// TwinCAT 3 PLC project SCARAFITTI
// ProgramVersion: 3.1.4023.0
// libraries:
//   Tc2_ControllerToolbox, * (Beckhoff Automation GmbH)
//   Tc2_Standard, * (Beckhoff Automation GmbH)
//   Tc2_System, * (Beckhoff Automation GmbH)
//   Tc2_Utilities, * (Beckhoff Automation GmbH)
//   Tc3_Module, * (Beckhoff Automation GmbH)
//   VisuSymbols,3.5.10.0,System
// project tree:
//   / GlobalTextList.TcGTLO, PlcTask.TcTTO, FastTask.TcTTO
//   GVLs/ Diagrama.TcCD (not stored), Cilindro.TcDUT, GVL.TcGVL, IO.TcGVL, SCARAFITTI.TcDUT
//   POUs/Actuadores/ PWM_valvulas.TcPOU (not stored)
//   POUs/Comunicacion/ EjecutarComando.TcPOU, G_buscar_numero.TcPOU, InterpretarComando.TcPOU, LetraPresente.TcPOU
//   POUs/ FB_BARRIDOXY.TcPOU, FB_SOLVEABCDE.TcPOU, FB_SOLVEALFABETA.TcPOU, MAIN.TcPOU, Simulacion.TcPOU
//   POUs/Functions/ TwoPiCrop.TcPOU
//   POUs/Sensores/ EncoderMeas.TcPOU, ENCODERPULSEtoANGLE.TcPOU
// real-time tasks:
//   TASK PlcTask: cycle T#10ms, priority 20, ADS port 350
//   TASK FastTask: cycle T#1ms, priority 1, ADS port 351
//   TASK VISU_TASK: cycle T#200000us, priority 30, ADS port 352
// I/O:
//   DEVICE Device 1 (EtherCAT) (disabled), AmsNetId 172.17.69.129.2.1
//     Term 7 (EK1200) [EK1200-5000 EtherCAT Power supply (2A E-Bus)]
//       Term 8 (EL1004) [EL1004 4Ch. Dig. Input 24V, 3ms]
//       Term 9 (EL1004) [EL1004 4Ch. Dig. Input 24V, 3ms]
//       Term 10 (EL2004) [EL2004 4Ch. Dig. Output 24V, 0.5A]
//       Term 11 (EL2004) [EL2004 4Ch. Dig. Output 24V, 0.5A]
//       Term 13 (EL9011) [EL9011 End Terminal]
// variable links:
//   SCARAFITTI/SCARAFITTI Instance <-> Device 1 (EtherCAT)/Term 7 (EK1200)/Term 10 (EL2004)
//     FastTask Outputs/IO.valv_alfa_mas <-> Channel 1/Output
//     FastTask Outputs/IO.valv_alfa_menos <-> Channel 2/Output
//     FastTask Outputs/IO.valv_beta_mas <-> Channel 3/Output
//     FastTask Outputs/IO.valv_beta_menos <-> Channel 4/Output
//   SCARAFITTI/SCARAFITTI Instance <-> Device 1 (EtherCAT)/Term 7 (EK1200)/Term 9 (EL1004)
//     FastTask Inputs/IO.encoder1_A <-> Channel 1/Input
//     FastTask Inputs/IO.encoder1_B <-> Channel 2/Input

CONFIGURATION SCARAFITTI
    RESOURCE PLC ON TwinCAT3
        TASK PlcTask(INTERVAL := T#10ms, PRIORITY := 20);
        TASK FastTask(INTERVAL := T#1ms, PRIORITY := 1);
        PROGRAM MAIN WITH PlcTask : MAIN;
        PROGRAM Simulacion WITH PlcTask : Simulacion;
        PROGRAM EncoderMeas WITH FastTask : EncoderMeas;
        PROGRAM PWM_valvulas WITH FastTask : PWM_valvulas;
        PROGRAM Simulacion WITH FastTask : Simulacion;
    END_RESOURCE
END_CONFIGURATION

// ---- GVLs/Cilindro.TcDUT
TYPE Cilindro :
STRUCT
	posicion : REAL;
	extendido: BOOL;
	retraido: BOOL;
	parado: BOOL;
	extendiendo : BOOL;
	retrayendo: BOOL;
	regimen : REAL; //tnato por uno de apertura de válvula
END_STRUCT
END_TYPE

// ---- GVLs/SCARAFITTI.TcDUT
TYPE SCARAFITTI :
STRUCT
	parada : BOOL;
	simulacion_alfa : BOOL;
	simulacion_beta : BOOL;
	quieto : BOOL;
	en_objetivo : BOOL;
	error_objetivo : BOOL;
	ADSCOM_ready : BOOL;
END_STRUCT
END_TYPE

// ---- GVLs/GVL.TcGVL
{attribute 'qualified_only'}
VAR_GLOBAL


// Geometría del robot//
//todo en mm//

Pi : REAL := 3.1416;

d : REAL := 400;
l1 : REAL := 1000; //longitud brazo proximal
l2 : REAL := 1400; //longitud brazo distal

//Vértices robot

Xa : REAL:= 0; 
Ya : REAL:= 0; 
Xb : REAL:= 0; 
Yb : REAL:= 0; 
Xc : REAL:= 0; //posición x del spray
Xc_sp : REAL:= 0; //setpoint posición x del spray
Yc : REAL:= 0; //posición y del spray
Yc_sp : REAL:= 0; //setpoint posición y del spray
Xd : REAL:= 0; 
Yd : REAL:= 0; 
Xe : REAL:= 0; 
Ye : REAL:= 0; 

//Mitad de cada brazo

Xab : REAL:= 0; 
Yab : REAL:= 0; 
Xbc : REAL:= 0; 
Ybc : REAL:= 0; 
Xcd : REAL:= 0; 
Ycd : REAL:= 0; 
Xde : REAL:= 0; 
Yde : REAL:= 0;


//Ángulos

alfa : REAL:= 0; //ángulo del brazo proximal izquierdo
alfa_sp : REAL:= 0; //setpoint ángulo del brazo proximal izquierdo
beta : REAL:= 0; //ángulo del brazo proximal derecho
beta_sp: REAL:= 0; //setpoint ángulo del brazo proximal derecho

deadband_angulo : REAL:= 0.05; //banda de no actuación en torno a target [rad]

alfa1 : REAL:= 0; 
beta1 : REAL:= 0; 
alfa2 : REAL:= 0; 
beta2 : REAL:= 0; 


d1: REAL;
d2: REAL;


alfa_enc : REAL :=0;
beta_enc : REAL :=0;

//cilindros
Cilindro1 : Cilindro;
Cilindro2 : Cilindro;
regimen_maximo : REAL :=100;

//Internas
en_objetivo_alfa : BOOL; //brazo proximal izquierdo en posición objetivo
en_objetivo_beta : BOOL; ///brazo proximal derecho en posición objetivo
comando_actual : STRING := 'Default comando actual';
ultimo_comando : STRING;
comando_actual_tipo : STRING;

//Sistema
Scarafitti : SCARAFITTI;

END_VAR

// ---- GVLs/IO.TcGVL
{attribute 'qualified_only'}
VAR_GLOBAL
//INPUTS	
	encoder1_A AT %I* : BOOL;
	encoder1_B AT %I* : BOOL;
	encoder2_A AT %I* : BOOL;
	encoder2_B AT %I* : BOOL;
	tope_alfa AT %I* : BOOL;
	tope_beta AT %I* : BOOL;
	
// INPUTS SIMULACION
	alfa_sim : REAL:= GVL.Pi;
	beta_sim : REAL;
	
// INPUTS ADS
	string_in : STRING := 'Default command PC-PLC';
	string_out : STRING:= 'Default feedback PLC-PC';
	
//OUTPUTS	
	blink AT %Q* : BOOL := 1;
	valv_alfa_mas AT %Q* : BOOL;
	valv_alfa_menos AT %Q* : BOOL;
	valv_beta_mas AT %Q* : BOOL;
	valv_beta_menos AT %Q* : BOOL;	
	
//OUTPUTS ADS
	Xc_ADS : INT;
	Yc_ADS : INT;
	alfa_deg:REAL;
	beta_deg:REAL;
END_VAR

// ---- POUs/MAIN.TcPOU
PROGRAM MAIN
VAR
	
fb_solveAlfaBeta:FB_SOLVEALFABETA;
fb_solveABCDE:FB_SOLVEABCDE;
fb_barridoXY:FB_BARRIDOXY;
InterpretarComando : InterpretarComando;
EjecutarComando: EjecutarComando;




Xc_test : LINT;
aux_ADS : INT;
Yc_test : LINT;

//test
nVar: UDINT;
//test
aux_UDINT : UDINT;
aux_REAL : REAL;

END_VAR

//Blink
IO.blink := NOT(IO.blink);


//DÓNDE ESTOY?
///comunicar ángulos
IO.alfa_deg:=GVL.alfa*180/GVL.Pi;
IO.beta_deg:=GVL.beta*180/GVL.Pi;
///Resolver geometría
////SolveABCDE
fb_solveABCDE.alfa:=GVL.alfa;
fb_solveABCDE.beta:=GVL.beta;
fb_solveABCDE();
GVL.Xa:=(fb_solveABCDE.Xa);
GVL.Ya:=(fb_solveABCDE.Ya);
GVL.Xb:=(fb_solveABCDE.Xb);
GVL.Yb:=(fb_solveABCDE.Yb);
GVL.Xc:=(fb_solveABCDE.Xc);
IO.Xc_ADS:=REAL_TO_INT(GVL.Xc);
IO.Yc_ADS:=REAL_TO_INT(GVL.Yc);
GVL.Yc:=(fb_solveABCDE.Yc);
GVL.Xd:=(fb_solveABCDE.Xd);
GVL.Yd:=(fb_solveABCDE.Yd);
GVL.Xe:=(fb_solveABCDE.Xe);
GVL.Ye:=(fb_solveABCDE.Ye);
////Brazos
GVL.Xab:=(GVL.Xa+GVL.Xb)/2;
GVL.Yab:=(GVL.Ya+GVL.Yb)/2;
GVL.Xbc:=(GVL.Xc+GVL.Xb)/2;
GVL.Ybc:=(GVL.Yc+GVL.Yb)/2;
GVL.Xcd:=(GVL.Xc+GVL.Xd)/2;
GVL.Ycd:=(GVL.Yc+GVL.Yd)/2;
GVL.Xde:=(GVL.Xd+GVL.Xe)/2;
GVL.Yde:=(GVL.Yd+GVL.Ye)/2;

//ADÓNDE VOY?
///Consigna XcYc
////Barrido para test
//fb_barridoXY.speed:=2;
//fb_barridoXY();
//GVL.Xc_sp:=fb_barridoXY.Xbarrido;
//GVL.Yc_sp:=fb_barridoXY.Ybarrido;
////ADS Com
IF ((NOT(GVL.Scarafitti.parada) AND GVL.Scarafitti.ADSCOM_ready AND IO.string_in<>GVL.ultimo_comando)OR IO.string_in='reset') THEN
	InterpretarComando();
	ELSE
		////Ignorar comandos que llegan mientras ADS com no está listo
		IO.string_in:=GVL.ultimo_comando;
END_IF

	

////Fija
//GVL.Xc_sp:= Xc_test;
//GVL.Yc_sp:= Yc_test;
///SolveAlfaBeta_sp
fb_solveAlfaBeta.x:=GVL.Xc_sp;
fb_solveAlfaBeta.y:=GVL.Yc_sp;
fb_solveAlfaBeta();
GVL.d1 :=fb_solveAlfaBeta.d1;
GVL.d2 :=fb_solveAlfaBeta.d2;
GVL.Scarafitti.error_objetivo := fb_solveAlfaBeta.error;
GVL.alfa_sp:=MIN(MAX(gvl.pi/2,fb_solveAlfaBeta.alfa),GVL.Pi);
GVL.beta_sp:=MIN(MAX(0,fb_solveAlfaBeta.beta),GVL.Pi/2);

//HE LLEGADO?
GVL.en_objetivo_alfa:=(ABS(GVL.alfa-GVL.alfa_sp)<=GVL.deadband_angulo);
GVL.en_objetivo_beta:=(ABS(GVL.beta-GVL.beta_sp)<=GVL.deadband_angulo);
GVL.Scarafitti.en_objetivo := GVL.en_objetivo_alfa AND GVL.en_objetivo_beta;


//SI NO HE LLEGADO, ME MUEVO
///si no hay parada
EjecutarComando();

END_PROGRAM

// ---- POUs/FB_SOLVEALFABETA.TcPOU
FUNCTION_BLOCK FB_SOLVEALFABETA
VAR_INPUT
x : REAL;
y : REAL;
END_VAR
VAR_OUTPUT
alfa : REAL;
beta : REAL;
d1 : REAL;
d2 : REAL;
alfa1 : REAL;
alfa2 : REAL;
beta1 : REAL;
beta2 : REAL;
error: BOOL := 0;

END_VAR
VAR
END_VAR

error:=FALSE;
d1 := SQRT(y*y+(x+GVL.d)*(x+GVL.d));
IF d1>(GVL.l1*GVL.l1+GVL.l2*GVL.l2) THEN
	error:=TRUE;
END_IF
d2 := SQRT(y*y+(x-GVL.d)*(x-GVL.d));
IF d2>(GVL.l1*GVL.l1+GVL.l2*GVL.l2) THEN
	error:=TRUE;
END_IF

IF (x+GVL.d=0) THEN
	alfa1:=GVL.Pi/2;
	ELSE IF x+GVL.d<0 THEN		
		alfa1 := gvl.pi + ATAN (y/(x+GVL.d));
		ELSE
			alfa1 := ATAN (y/(x+GVL.d));
		END_IF
	END_IF
IF alfa1 < 0 THEN
	error:=TRUE;
END_IF

IF (x-GVL.d=0) THEN
	beta1:=GVL.Pi/2;
	ELSE IF x-GVL.d>0 THEN
		beta1 := ATAN (y/(x-GVL.d));
	ELSE
		beta1 := GVL.Pi	+ ATAN (y/(x-GVL.d));
	END_IF
	END_IF

IF beta1 < 0 THEN
	error:=TRUE;
END_IF

IF (ABS((GVL.l1*GVL.l1+d1*d1-GVL.l2*GVL.l2)/(2*GVL.l1*d1))>1) THEN
error := TRUE;
END_IF

IF (ABS((GVL.l1*GVL.l1+d2*d2-GVL.l2*GVL.l2)/(2*GVL.l1*d2))>1) THEN
error := TRUE;
END_IF

IF error=FALSE THEN
	IF d1=0 THEN
		alfa2:=0;
		ELSE
			alfa2 := ABS(ACOS((GVL.l1*GVL.l1+d1*d1-GVL.l2*GVL.l2)/(2*GVL.l1*d1)));
		END_IF

	
	IF d2=0 THEN
		beta2:=0;
		ELSE
			beta2 := ABS(ACOS((GVL.l1*GVL.l1+d2*d2-GVL.l2*GVL.l2)/(2*GVL.l1*d2)));
		END_IF
alfa := alfa1 + alfa2;
beta := beta1 - beta2;
	END_IF

END_FUNCTION_BLOCK

// ---- POUs/FB_SOLVEABCDE.TcPOU
FUNCTION_BLOCK FB_SOLVEABCDE
VAR_INPUT
	alfa : REAL:= 0; //ángulo del brazo pxosimal izquierdo
	beta : REAL:= 0; //ángulo del brazo pxosimal derecho
END_VAR
VAR_OUTPUT
	
	Xa : REAL:= 0; 
	Ya : REAL:= 0; 
	Xb : REAL:= 0; 
	Yb : REAL:= 0; 
	Xc : REAL:= 0; 
	Yc : REAL:= 0;
	Xd : REAL:= 0; 
	Yd : REAL:= 0; 
	Xe : REAL:= 0; 
	Ye : REAL:= 0; 
	error : BOOL :=0;
	check_AB : REAL:=GVL.l1;
	check_BC : REAL:=GVL.l2;
	check_CD : REAL:=GVL.l2;
	check_DE : REAL:=GVL.l1;
	

END_VAR
VAR
	aux1 : REAL;
	aux2 : REAL;
	A : REAL;
	B : REAL;
	C : REAL;
END_VAR

error:=FALSE;

// A
Xa := -GVL.d ;
Ya := 0 ;

//B
Xb := Xa + GVL.l1*COS(alfa);
Yb := GVL.l1*SIN(alfa);

//E
Xe := GVL.d ;
Ye := 0 ;

//D
Xd := Xe + GVL.l1*COS(beta);
Yd := GVL.l1*SIN(beta);

//Chekcs
IF SQRT((Xd-Xb)*(Xd-Xb)+(Yd-Yb)*(Yd-Yb))>2*GVL.l2 THEN //B y D demaisado separados
	error:=TRUE;
	ELSE IF Xb>=Xd THEN //brazos proximales cruzados
		error:=TRUE;
		ELSE //calculate Xc
			aux1:=(Xb*Xb-Xd*Xd+Yb*Yb-Yd*Yd)/(2*(Xb-Xd));
			aux2:=-(Yb-Yd)/(Xb-Xd);
			A:=1+ aux2*aux2 ;
			B:=2*(aux1*aux2-Xb*aux2-Yb);
			C:=aux1*aux1-2*Xb*aux1+Yb*Yb+Xb*Xb-GVL.l2*GVL.l2;
			Yc := (-B+SQRT(B*B-4*A*C))/(2*A);
			Xc := aux1+aux2*Yc;
		END_IF
		
check_AB:=SQRT((Xb-Xa)*(Xb-Xa)+(Yb-Ya)*(Yb-Ya));
check_BC:=SQRT((Xb-Xc)*(Xb-Xc)+(Yb-Yc)*(Yb-Yc));
check_CD:=SQRT((Xd-Xc)*(Xd-Xc)+(Yd-Yc)*(Yd-Yc));
check_DE:=SQRT((Xd-Xe)*(Xd-Xe)+(Yd-Ye)*(Yd-Ye));
		
	END_IF

END_FUNCTION_BLOCK

// ---- POUs/FB_BARRIDOXY.TcPOU
FUNCTION_BLOCK FB_BARRIDOXY
VAR_INPUT
	speed : REAL;
END_VAR
VAR_OUTPUT
	Xbarrido: REAL := 0;
	Ybarrido : REAL :=1000;
END_VAR
VAR
	xmax : REAL := 500;
	ymin : REAL := 500;
	ymax : REAL := 1500;
	fase : INT := 1;
END_VAR

CASE fase OF
	1:
	IF Xbarrido + speed > xmax THEN
		fase:=2;
		ELSE
			Xbarrido := Xbarrido + speed;
	END_IF
	2:
	IF Ybarrido + speed > ymax THEN
		fase:=3;
		ELSE
			Ybarrido := Ybarrido + speed;
	END_IF
	3:
	IF Xbarrido - speed < -xmax THEN
		fase:=4;
		ELSE
			Xbarrido := Xbarrido - speed;
	END_IF
	4:
	IF Ybarrido - speed < ymin THEN
		fase:=1;
		ELSE
			Ybarrido := Ybarrido - speed;
	END_IF
END_CASE

END_FUNCTION_BLOCK

// ---- POUs/Comunicacion/InterpretarComando.TcPOU
FUNCTION_BLOCK InterpretarComando
VAR_INPUT
END_VAR
VAR_OUTPUT
	comando_valido:BOOL;
END_VAR
VAR
	aux_str:STRING;
	aux_int:INT;
	aux_real:REAL;
	buscarX:G_buscar_numero;
	buscarY:G_buscar_numero;
	buscarF:G_buscar_numero;
	buscarS:G_buscar_numero;
	
END_VAR

comando_valido:=FALSE;
///Comando en mayúsculas
IO.string_in:=f_toucase(IO.string_in);
///excepcion para reset
IF IO.string_in='RESET' THEN
	IO.string_in:='G00 X000 Y000';
END_IF
	IF  letraPresente('G',IO.string_in) THEN
		IF letraPresente('G00',IO.string_in) THEN
			IO.string_out:='comando G00 recibido';
			//buscar comandos de X
			IF letraPresente('X',IO.string_in) THEN
			buscarX.cadena:=IO.string_in;
			buscarX.letra:='X';
			buscarX();
			GVL.Xc_sp:= buscarX.numero;
			GVL.comando_actual:=IO.string_in;
			GVL.comando_actual_tipo:='G00';
			GVL.Scarafitti.ADSCOM_ready:=FALSE;
			comando_valido:=TRUE;
			END_IF
			//buscar comandos de Y
			IF letraPresente('Y',IO.string_in) THEN
			buscarY.cadena:=IO.string_in;
			buscarY.letra:='Y';
			buscarY();
			GVL.Yc_sp:= buscarY.numero;
			GVL.comando_actual:=IO.string_in;
			GVL.comando_actual_tipo:='G00';
			GVL.Scarafitti.ADSCOM_ready:=FALSE;
			comando_valido:=TRUE;
			END_IF
			
		ELSE IF letraPresente('G01',IO.string_in) THEN
			IO.string_out:='comando G01 recibido';
			//buscar comandos de X
			IF letraPresente('X',IO.string_in) THEN
			buscarX.cadena:=IO.string_in;
			buscarX.letra:='X';
			buscarX();
			GVL.Xc_sp:= buscarX.numero;
			GVL.comando_actual:=IO.string_in;
			GVL.comando_actual_tipo:='G01';
			GVL.Scarafitti.ADSCOM_ready:=FALSE;
			comando_valido:=TRUE;
			END_IF
			//buscar comandos de Y
			IF letraPresente('Y',IO.string_in) THEN
			buscarY.cadena:=IO.string_in;
			buscarY.letra:='Y';
			buscarY();
			GVL.Yc_sp:= buscarY.numero;
			GVL.comando_actual:=IO.string_in;
			GVL.comando_actual_tipo:='G01';
			GVL.Scarafitti.ADSCOM_ready:=FALSE;
			comando_valido:=TRUE;
			END_IF
			END_IF
			END_IF
END_IF
	///buscar comandos F de velocidad
	IF letraPresente('F',IO.string_in) THEN
			buscarF.cadena:=IO.string_in;
			buscarF.letra:='F';
			buscarF();
			GVL.regimen_maximo:= buscarF.numero;
			comando_valido:=TRUE;
		END_IF

//comando desconocido
IF NOT(letraPresente('G',IO.string_in) OR letraPresente('F',IO.string_in)) THEN
	 IO.string_out:='Comando desconocido';
		GVL.comando_actual:='Comando desconocido';
		GVL.Scarafitti.ADSCOM_ready:=TRUE;
	END_IF

//actualizar último comando sólo si es válido
IF comando_valido THEN
	GVL.ultimo_comando:=IO.string_in;
END_IF

END_FUNCTION_BLOCK

// ---- POUs/Comunicacion/G_buscar_numero.TcPOU
FUNCTION_BLOCK G_buscar_numero
VAR_INPUT
	letra : STRING;
	cadena : STRING;
	
END_VAR
VAR_OUTPUT
	numero : REAL;
	error:BOOL;
END_VAR
VAR
	aux:INT;
	inicio:INT;
	espacio_siguiente:INT;
	cadena_recortada:STRING;
END_VAR

error:=FALSE;
numero:=0.99;
IF find(cadena,letra)=0 THEN
	error:=TRUE;
	ELSE
		aux:=find(cadena,letra);
		inicio:=aux + 1;
		cadena_recortada:=delete(cadena,aux,1);
		espacio_siguiente:=find(cadena_recortada,' ');
		IF espacio_siguiente=0 THEN
			espacio_siguiente := len(cadena_recortada)+1;
		END_IF
		numero:=STRING_TO_REAL(left(cadena_recortada,espacio_siguiente -1));
END_IF

END_FUNCTION_BLOCK

// ---- POUs/Comunicacion/LetraPresente.TcPOU
FUNCTION LetraPresente : BOOL
VAR_INPUT
	letra: STRING;
	cadena: STRING;
END_VAR
VAR
END_VAR

LetraPresente := FIND (cadena,letra) > 0;

END_FUNCTION

// ---- POUs/Comunicacion/EjecutarComando.TcPOU
FUNCTION_BLOCK EjecutarComando
VAR_INPUT
END_VAR
VAR_OUTPUT
END_VAR
VAR
	dalfa : REAL;
	dbeta : REAL;
END_VAR

IF NOT(GVL.Scarafitti.parada) THEN 
	IF GVL.comando_actual_tipo='G00' THEN
		///inicializar regimenes a cero
		GVL.Cilindro1.regimen:=0;
		GVL.Cilindro2.regimen:=0;
		IF NOT GVL.en_objetivo_alfa THEN
	IF GVL.alfa<GVL.alfa_sp THEN
		GVL.Cilindro1.regimen:=GVL.regimen_maximo;
		ELSE IF GVL.alfa>GVL.alfa_sp THEN
		GVL.Cilindro1.regimen:=-GVL.regimen_maximo;
	END_IF
END_IF
END_IF
IF NOT GVL.en_objetivo_beta THEN
	IF GVL.beta<GVL.beta_sp THEN
		GVL.Cilindro2.regimen:=GVL.regimen_maximo;
		ELSE IF GVL.beta>GVL.beta_sp THEN
		GVL.Cilindro2.regimen:=-GVL.regimen_maximo;
	END_IF
END_IF
END_IF
	ELSE IF GVL.comando_actual_tipo='G01' THEN
		///inicializar regimenes a cero
		GVL.Cilindro1.regimen:=0;
		GVL.Cilindro2.regimen:=0;
		IF NOT GVL.Scarafitti.en_objetivo THEN
		///determinar la diferencia con el objetivo en alfa y beta
		dalfa:=GVL.alfa_sp-GVL.alfa;
		dbeta:=GVL.beta_sp-GVL.beta;
		//si alfa está más lejos que beta
		IF ABS(dalfa)>ABS(dbeta) THEN
			IF NOT GVL.en_objetivo_alfa THEN
			IF dalfa > 0 THEN
				//mover cilindro 1 a velocidad máxima
				GVL.Cilindro1.regimen:=GVL.regimen_maximo;
				ELSE
					//o mínima
					GVL.Cilindro1.regimen:=-GVL.regimen_maximo;
				END_IF
			END_IF
				//y mover cilindro 2 a menor velocidad dbeta/dalfa
			IF NOT GVL.en_objetivo_beta THEN
				IF dbeta >0 THEN
					GVL.Cilindro2.regimen:=GVL.regimen_maximo*ABS(dbeta/dalfa);
					ELSE
						GVL.Cilindro2.regimen:=-GVL.regimen_maximo*ABS(dbeta/dalfa);
					END_IF
			END_IF

			// si beta está más lejos que alfa
			ELSE
			IF NOT GVL.en_objetivo_beta THEN
			IF dbeta > 0 THEN
				//mover cilindro 2 a velocidad máxima
				GVL.Cilindro2.regimen:=GVL.regimen_maximo;
				ELSE
					//o mínima
					GVL.Cilindro2.regimen:=-GVL.regimen_maximo;
				END_IF
			END_IF
				//y mover cilindro 1 a menor velocidad dalfa/dbeta
			IF NOT GVL.en_objetivo_alfa THEN
				IF dalfa >0 THEN
					GVL.Cilindro1.regimen:=GVL.regimen_maximo*ABS(dalfa/dbeta);
					ELSE
						GVL.Cilindro1.regimen:=-GVL.regimen_maximo*ABS(dalfa/dbeta);
					END_IF
			END_IF
			END_IF
		
		END_IF
	END_IF
	END_IF
				END_IF
	
//SI NO HE LLEGADO NO ACEPTO NUEVO COMANDO
IF NOT GVL.Scarafitti.en_objetivo THEN
	GVL.Scarafitti.ADSCOM_ready := FALSE;
	IO.string_out := CONCAT('Executing: ',gvl.comando_actual);
	ELSE
		GVL.Scarafitti.ADSCOM_ready := TRUE;
		IO.string_out := concat(concat(concat(CONCAT( 'Ready at Xc=', INT_TO_STRING(IO.Xc_ADS)), 'mm, Yc='),  INT_TO_STRING(IO.Yc_ADS)) , 'mm');
END_IF

//SI EL SETPOINT ES ERRONEO, AVISAR Y ABRIR CANAL
IF GVL.Scarafitti.error_objetivo THEN
		GVL.Scarafitti.ADSCOM_ready := TRUE;
		IO.string_out := 'Objetivo inválido, mandar nuevo comando';
END_IF

//SI EL COMANDO ES DESCONOCIDO, AVISAR Y ABRIR CANAL

IF GVL.comando_actual='Comando desconocido' THEN
			GVL.Scarafitti.ADSCOM_ready := TRUE;
		IO.string_out := 'Comando desconocido, mandar nuevo comando';
END_IF

END_FUNCTION_BLOCK

// ---- POUs/Simulacion.TcPOU
PROGRAM Simulacion
VAR
	vel : REAL := 0.001;

END_VAR

//nuevos ángulos
IF IO.valv_alfa_mas THEN
	IO.alfa_sim:=IO.alfa_sim + vel;
	ELSE IF IO.valv_alfa_menos THEN
		IO.alfa_sim := (IO.alfa_sim - vel);
	END_IF

END_IF

IF IO.valv_beta_mas THEN
	IO.beta_sim:=IO.beta_sim + vel;
	ELSE IF IO.valv_beta_menos THEN
		IO.beta_sim := IO.beta_sim - vel;
	END_IF

END_IF

IO.alfa_sim:=TwoPiCrop(IO.alfa_sim);
IO.beta_sim:=TwoPiCrop(IO.beta_sim);

END_PROGRAM

// ---- POUs/Functions/TwoPiCrop.TcPOU
FUNCTION TwoPiCrop : REAL
VAR_INPUT
	in:REAL;
END_VAR
VAR
	aux_LINT:LINT;
END_VAR

aux_LINT:=REAL_TO_LINT(in*1000000);
aux_LINT:= aux_LINT MOD REAL_TO_LINT(1000000*2*GVL.Pi);
TwoPiCrop:= LINT_TO_REAL(aux_LINT)/1000000;
IF TwoPiCrop < 0 THEN
	TwoPiCrop := 2*GVL.Pi - TwoPiCrop;
END_IF

END_FUNCTION

// ---- POUs/Sensores/EncoderMeas.TcPOU
PROGRAM EncoderMeas
VAR
	
encoder1:ENCODERPULSEtoANGLE;
encoder2:ENCODERPULSEtoANGLE;

END_VAR

//Dónde estoy?

//ALFA
///Realidad
IF NOT(GVL.Scarafitti.simulacion_alfa) THEN
////Calibración
encoder1.angulo_calibrado:=GVL.Pi;
encoder1.b_calibrado:=IO.tope_alfa;
////Medir ángulos
encoder1.A:=IO.encoder1_A;
encoder1.B:=IO.encoder1_B;
encoder1();
GVL.alfa:=encoder1.angle;
ELSE
///Simulación
GVL.alfa:=IO.alfa_sim;
END_IF

//BETA
///Realidad
IF NOT(GVL.Scarafitti.simulacion_beta) THEN
////Calibración
encoder2.angulo_calibrado:=0;
encoder2.b_calibrado:=IO.tope_beta;
////Medir ángulos
encoder2.A:=IO.encoder2_A;
encoder2.B:=IO.encoder2_B;
encoder2();
GVL.beta:=encoder2.angle;
ELSE
///Simulación
GVL.beta:=IO.beta_sim;
END_IF

END_PROGRAM

// ---- POUs/Sensores/ENCODERPULSEtoANGLE.TcPOU
FUNCTION_BLOCK ENCODERPULSEtoANGLE
VAR_INPUT
	A :BOOL;
	B:BOOL;
	Pulsos:DINT:=1600;
	b_calibrado: BOOL;
	angulo_calibrado : REAL;
END_VAR
VAR_OUTPUT
	acum : DINT:=0;
	angle :REAL;
	estado : INT;
END_VAR
VAR
	delta_angulo : REAL;
END_VAR

//determinar delta angulo
delta_angulo:=2*GVL.pi/pulsos;

//ACUM
CASE estado OF
	0: //INIT
	IF(A AND NOT(B)) THEN
		estado:=1;
		ELSE IF A AND B THEN
			estado:=2;
			ELSE IF B AND NOT(A) THEN
				estado:=3;
				ELSE IF NOT(B)AND NOT(A) THEN
					estado:=4;
				END_IF
			END_IF
			
		END_IF
	END_IF
	estado:=1;
	1:
	IF B THEN
		estado:=2;
		acum:=acum+1;
		angle:=angle + delta_angulo;
		ELSE IF NOT(A) THEN
			estado:=4;
			acum:=acum-1;
			angle:=angle - delta_angulo;
		END_IF
	END_IF
	2:
	IF NOT(A) THEN
		estado:=3;
		acum:=acum+1;
		angle:=angle + delta_angulo;
		ELSE IF NOT(B) THEN
			estado:=1;
			acum:=acum-1;
			angle:=angle - delta_angulo;
		END_IF
	END_IF
	3:
	IF NOT(B) THEN
		estado:=4;
		acum:=acum+1;
		angle:=angle + delta_angulo;
		ELSE IF A THEN
			estado:=2;
			acum:=acum-1;
			angle:=angle - delta_angulo;
		END_IF
	END_IF
	4:
	IF A THEN
		estado:=1;
		acum:=acum+1;
		angle:=angle + delta_angulo;
		ELSE IF B THEN
			estado:=3;
			acum:=acum-1;
			angle:=angle - delta_angulo;
		END_IF
	END_IF
	
END_CASE

//calibración
IF b_calibrado THEN
	acum:=0;
	angle:=angulo_calibrado;	
END_IF

END_FUNCTION_BLOCK

// ---- GlobalTextList.TcGTLO
TEXTLIST GlobalTextList
  281 = '+'
  249 = '-'
  933 = 'ALFA'
  513 = 'BETA'
  70 = 'PARADA'
  719 = 'REGIMEN MAXIMO'
  276 = 'SIMULACION'
  526 = 'STATUS'
END_TEXTLIST
